// TIA Portal V19 export
TYPE "C301_VAR_CLUST_TYPIC"
   STRUCT
      CAPA_OK { ExternalAccessible := 'False'; ExternalVisible := 'False'; ExternalWritable := 'False'} : USInt;   // Aantal bestuurbare ventilatoren in de cluster
      NIV_AAN_BWA { ExternalAccessible := 'False'; ExternalVisible := 'False'; ExternalWritable := 'False'} : USInt;   // Aantal aangeschakelde ventilatoren in de gewenste ventilatierichting
      DIR { ExternalAccessible := 'False'; ExternalVisible := 'False'; ExternalWritable := 'False'} : USInt;   // Richting van de cluster
      BMO { ExternalAccessible := 'False'; ExternalVisible := 'False'; ExternalWritable := 'False'} : USInt;   // Bedieningsmode
      ONHD_STS { ExternalAccessible := 'False'; ExternalVisible := 'False'; ExternalWritable := 'False'} : USInt;   // Status automatische onderhoudstesten
      PWR { ExternalAccessible := 'False'; ExternalVisible := 'False'; ExternalWritable := 'False'} : Real;   // Actueel vermogen van de ventilatiecluster
   END_STRUCT;
END_TYPE
